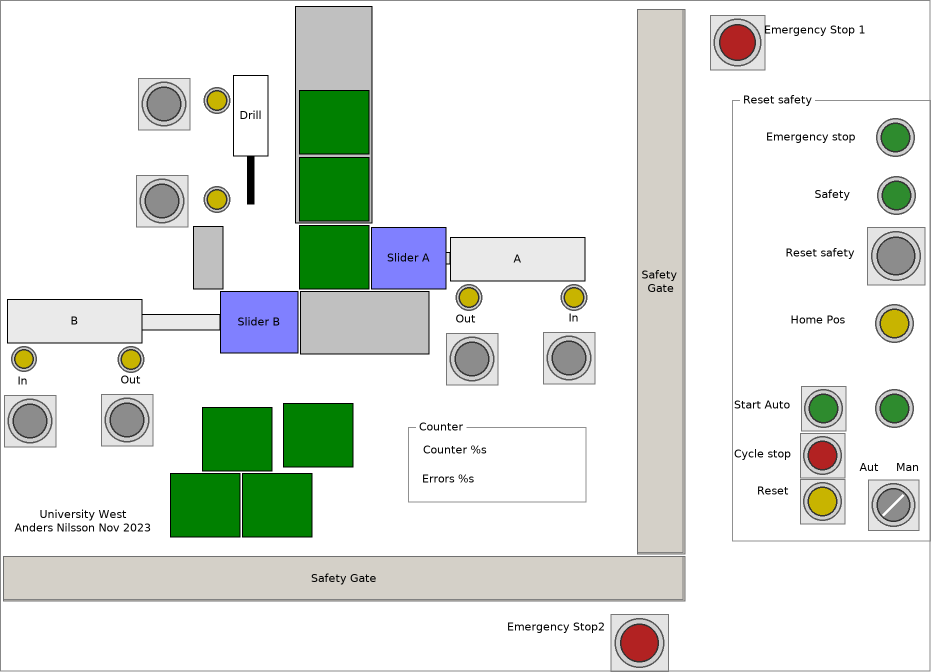
VISUALIZATION Visualization  // 931x672
    Group (233,75 59x138)
        p2773130477: main.nPosDrill
        p1126004900: MAIN.nPosDrill
        Rectangle (0,0 35x81), "Drill"
        Rectangle (14,81 7x48)
    Rectangle (295,6 77x217)
    Rectangle (299,225 70x64), invisible if: MAIN.mxCubeInvisible
        p3528305787: MAIN.nPosXCube
        p874137650: MAIN.nPosXCube
        p2773130477: MAIN.nPosYCube
        p1126004900: MAIN.nPosYCube
    Rectangle (193,226 30x63)
    Rectangle (299,157 70x64)
    Rectangle (300,291 129x63)
    Rectangle (299,90 70x64)
    Lamp1 (115,344 32x31), variable: MAIN.qxSliderBout, style: Lamp-Lamp1-Yellow
    Lamp1 (8,344 32x30), variable: MAIN.qxSliderBin, style: Lamp-Lamp1-Yellow
    Lamp1 (558,282 32x31), variable: MAIN.qxSliderAin, style: Lamp-Lamp1-Yellow
    Lamp1 (453,282 32x31), variable: MAIN.qxSliderAout, style: Lamp-Lamp1-Yellow
    Lamp1 (201,85 32x31), variable: MAIN.qxDrillUp, style: Lamp-Lamp1-Yellow
    Lamp1 (201,184 32x31), variable: MAIN.qxDrillDown, style: Lamp-Lamp1-Yellow
    Rectangle (242,473 70x64), invisible if: main.nCnt < 1
    Rectangle (283,403 70x64), invisible if: main.nCnt < 4
    Rectangle (170,473 70x64), invisible if: main.nCnt < 2
    Rectangle (202,407 70x64), invisible if: main.nCnt < 3
    GroupBox (732,92 199x449), "Reset safety"
        Label (0,290 60x46), "Start Auto"
        PushSwitch (69,294 45x45), variable: MAIN.qxButtonStart, behaviour: TAP, style: Switch-PushSwitch-Green
        PushSwitch (68,341 45x45), variable: MAIN.qxButtonStop, behaviour: TAP, style: Switch-PushSwitch-Red
        Lamp1 (140,294 45x45), variable: MAIN.ixLampStarted, style: Lamp-Lamp1-Green
        Label (0,339 61x46), "Cycle stop"
        Label (50,133 76x56), "Reset safety"
        PushSwitch (135,134 58x60), variable: MAIN.qxBtnReset, behaviour: TAP, style: Switch-PushSwitch-Gray
        Label (75,88 51x29), "Safety"
        Label (32,17 94x56), "Emergency stop"
        Lamp1 (141,23 45x45), variable: MAIN.ixLampEmStopOk, style: Lamp-Lamp1-Green
        Lamp1 (142,81 45x45), variable: MAIN.ixLampSafetyOk, style: Lamp-Lamp1-Green
        RotarySwitch (136,386 51x54), variable: MAIN.qxAuto, behaviour: TOGGLE, style: Switch-RotarySwitch-Gray
        Label (121,362 73x27), "Aut Man"
        Lamp1 (140,209 45x45), variable: MAIN.ixLampHomePos, style: Lamp-Lamp1-Yellow
        Label (48,200 76x56), "Home Pos"
        Label (20,376 42x46), "Reset"
        PushSwitch (68,387 45x45), variable: MAIN.mxReset, behaviour: TAP, style: Switch-PushSwitch-Yellow
    GroupBox (408,419 178x83), "Counter"
        Rectangle (12,16 112x30), "Counter %s", text variable: MAIN.nCnt
        Rectangle (11,45 112x30), "Errors %s", text variable: MAIN.nErrorCnt
    Label (447,302 37x34), "Out"
    Label (112,363 37x34), "Out"
    Label (555,301 37x34), "In"
    Label (4,364 37x34), "In"
    Rectangle (371,252 79x12)
    Rectangle (450,237 135x44), "A"
    Rectangle (139,314 81x16)
    Rectangle (7,299 135x44), "B"
    Rectangle (371,227 75x62), "Slider A"
        p3528305787: MAIN.nPosSliderA
        p874137650: MAIN.nPosSliderA
    Rectangle (220,291 78x62), "Slider B"
        p3528305787: MAIN.nPosSliderB
        p874137650: MAIN.nPosSliderB
    Label (7,500 152x42), "University West Anders Nilsson Nov 2023"
    PushSwitch (446,332 52x54), variable: MAIN.qxBtnAout, behaviour: TAP, style: Switch-PushSwitch-Gray
    PushSwitch (543,331 52x54), variable: MAIN.qxBtnAin, behaviour: TAP, style: Switch-PushSwitch-Gray
    PushSwitch (101,393 52x54), variable: MAIN.qxBtnBout, behaviour: TAP, style: Switch-PushSwitch-Gray
    PushSwitch (4,394 52x54), variable: MAIN.qxBtnBin, behaviour: TAP, style: Switch-PushSwitch-Gray
    PushSwitch (136,174 52x54), variable: MAIN.qxBtnDrillOut, behaviour: TAP, style: Switch-PushSwitch-Gray
    PushSwitch (138,77 52x54), variable: MAIN.qxBtnDrillIn, behaviour: TAP, style: Switch-PushSwitch-Gray
    PushSwitch (703,15 69x55), variable: MAIN.mxBtn1EmStop, behaviour: TOGGLE, style: Switch-PushSwitch-Red
    Button (637,9 48x545), "Safety Gate"
        toggle MAIN.qxSafety1StopOk
    PushSwitch (606,614 67x58), variable: MAIN.mxBtn2EmStop, behaviour: TOGGLE, style: Switch-PushSwitch-Red
    Button (3,556 682x45), "Safety Gate"
        toggle MAIN.qxSafety2StopOk
    Label (745,2 140x56), "Emergency Stop 1"
    Label (486,599 140x56), "Emergency Stop2"
END_VISUALIZATION

(* stored: Version 1.1.0.1
   Visu Visualization: Id {6a967cc4-b88c-4500-a7a1-abfc74b431c0} *)
